FUNCTION_BLOCK FB_Sequence
(*
    Canonical command sequence: PLCopen-style interface over a state machine.
    Copy this shape for anything with steps or waiting.

    Contract: call this FB unconditionally every cycle. bExecute is edge-triggered.
    Every waiting state has a timeout and a path to Error. Error is resettable.
*)
VAR_INPUT
    bExecute    : BOOL;                 // rising edge starts the sequence
    bReset      : BOOL;                 // clears the error state
    tStepTimeout: TIME := T#10S;        // max time allowed in any one step
END_VAR
VAR_OUTPUT
    bBusy       : BOOL;                 // sequence is running
    bDone       : BOOL;                 // completed successfully (until next Execute edge)
    bError      : BOOL;
    nErrorID    : UDINT;                // 0 = no error; see GVL_Errors
END_VAR
VAR
    eState      : E_SeqState := E_SeqState.Idle;
    fbExecTrig  : R_TRIG;
    fbStepTimer : TON;
END_VAR
VAR CONSTANT
    cErrStep1Timeout : UDINT := 16#8101;
    cErrStep2Timeout : UDINT := 16#8102;
    cErrInvalidState : UDINT := 16#8FFF;
END_VAR

// Rule 2: edge detector is an instance and is called every cycle.
fbExecTrig(CLK := bExecute);

// Reset is handled outside the state machine so it works from any state.
IF bReset AND eState = E_SeqState.Error THEN
    nErrorID := 0;
    eState   := E_SeqState.Idle;
END_IF

CASE eState OF

    E_SeqState.Idle:
        IF fbExecTrig.Q THEN
            bDone  := FALSE;
            bError := FALSE;
            M_EnterStep(newState := E_SeqState.Step1);
        END_IF

    E_SeqState.Step1:
        // Rule 5: timer instance driven every cycle while in this state.
        fbStepTimer(IN := TRUE, PT := tStepTimeout);
        IF TRUE THEN                            // <- replace with the real step-1 done condition
            M_EnterStep(newState := E_SeqState.Step2);
        ELSIF fbStepTimer.Q THEN
            M_Fail(errorID := cErrStep1Timeout);
        END_IF

    E_SeqState.Step2:
        fbStepTimer(IN := TRUE, PT := tStepTimeout);
        IF TRUE THEN                            // <- replace with the real step-2 done condition
            M_EnterStep(newState := E_SeqState.Done);
        ELSIF fbStepTimer.Q THEN
            M_Fail(errorID := cErrStep2Timeout);
        END_IF

    E_SeqState.Done:
        bDone  := TRUE;
        eState := E_SeqState.Idle;

    E_SeqState.Error:
        // Define the safe output state here - what must be switched off on failure.
        ;

ELSE
    // Rule: an unreachable state means memory corruption or a missed CASE label.
    M_Fail(errorID := cErrInvalidState);
END_CASE

bBusy  := (eState <> E_SeqState.Idle) AND (eState <> E_SeqState.Error);
bError := (eState = E_SeqState.Error);

METHOD PRIVATE M_EnterStep
VAR_INPUT
    newState : E_SeqState;
END_VAR
// Reset the step timer on every transition so a re-entered state
// does not start with an already-elapsed timer (Rule 5).
fbStepTimer(IN := FALSE);
eState := newState;
END_METHOD

METHOD PRIVATE M_Fail
VAR_INPUT
    errorID : UDINT;
END_VAR
nErrorID := errorID;
fbStepTimer(IN := FALSE);
eState   := E_SeqState.Error;
END_METHOD

END_FUNCTION_BLOCK

(* stored: Version 1.1.0.1, ProductVersion 3.1.4024.0
   POU FB_Sequence: Id {f1de8ec9-179b-4df8-9097-158ff83ac1af}, SpecialFunc None
   Method M_EnterStep: Id {c2aa5b89-eee4-4849-8357-4bec2013ba32}
   Method M_Fail: Id {4df4ca21-902d-4af4-8bb4-b5dc09e5bd1d} *)
